// TIA Portal V16 export
// export: Created 2023-03-29T11:04:47.8257931Z, ExportSetting WithDefaults, DisplayName Totally Integrated Automation Portal, DisplayVersion V16 Update 6, DisplayName TIA Portal Version Control Interface, DisplayVersion V16 Update 2, DisplayName TIA Portal Openness, DisplayVersion V16 Update 6, DisplayName STEP 7 Professional, DisplayVersion V16 Update 6, DisplayName STEP 7 Safety, DisplayVersion V16, DisplayName WinCC Advanced, DisplayVersion V16 Update 6
FUNCTION_BLOCK "Sterowanie dołączeniem falownika"   // FB8, LAD
TITLE = Sterowanie dołączaniem styczników falownika
{ S7_Optimized_Access := 'TRUE' }
AUTHOR : rtecmer
VERSION : 0.1
// Sterowa stycznikiem pracy z falownika.
// Funkcja FB8 komutuje załaczenie stycznika FALOWNIK dla konkretnego napędu. Napędem sterowanym jest zawsze napęd przypisany do MC (czyli IsReady_MC to jest gotowość napędu sterowaniego) Na wejścia oznaczone wyróżnikiem MC podlączamy sygnały tej samej dmuchawy, której stycznikiem będziemy sterować poprzez wtjście setSUPV_FM
//  
// Sterowanie stycznikiem . Ustawianie znaczników setCMD_FM i setSUPV_FM które przekazywane są do funkcji FC3/FC1 DRV01 driver napędów. Następnie przekazywane jest do warstwy Hawtware/ OUT gdzie ustawiane jest wyjście sterownika
// stored: AutoNumber true, IsIECCheckEnabled false, IsRetainMemResEnabled false, MemoryReserve 500, SetENOAutomatically false, UDAEnableTagReadback false
   VAR_INPUT
      Is_up_Hz : Bool;
      Set_HWork_M : Bool;   // Znacznik ustawienia pracy od licznika
      setPID_Pompy : Bool;   // Znacznik załączenie, regulacji falownika
      IsRunInverter_MA : Bool;   // Potwierdzenie pracy z falownika kompresor dodatkowy 1
      IsRunNetwork_MA : Bool;   // Potwierdzenie praca z sieć dodatkowego
      IsRunInverter_MB : Bool;   // Potwierdzenie pracy z falownika kompresor dodatkowy 2
      IsRunNetwork_MB : Bool;   // Potwierdzenie praca z sieć dodatkowego
      IsRunNetwork_MC : Bool;   // Potwierdzenie pracy z sieci
      IsRunInverter_MC : Bool;   // Potwierdzenie pracy z falownika
      IsRunNetwork_MD : Bool;   // Potwierdzenie pracy z sieci
      IsRunInverter_MD : Bool;   // Potwierdzenie pracy z falownika
      FC2_Set_50H : Bool;   // Znacznik osiągnięcia czasu dla 50Hz
      IsRunInverter1 : Bool;   // Potwierdzenie pracy falownika / Potwierdzenie pracy falownika kompresorów M7M8M9
      AlwaysTRUE : Bool;
      IsReady_MA : Bool;   // Znacznik gotowości
      IsReady_MB : Bool;   // Znacznik gotowości
      IsReady_MC : Bool;   // Znacznik gotowości
      IsReady_MD : Bool;   // Znacznik gotowości
      IsModeAut : Bool;   // Znacznik trybu automat
      FB9_Set_Motor2 : Bool;   // Polecenie dostawienia dodatkowej nr1
      FB9_Set_Motor3 : Bool;   // Polecenie dostawienia dodatkowej nr2
      FB9_Set_Motor4 : Bool;   // Polecenie dostawienia dodatkowej nr3
      IsReady_Inverter : Bool;   // Gotowość falownika
      ResWorkInverter_to_MaxTime : Bool;   // Bit kasowania pracy falownika od maxymalnej ciągłej pracy
   END_VAR
   VAR_OUTPUT
      setSUPV_FM : Bool;   // Znacznik polecenia startu z falownika
   END_VAR
   VAR_IN_OUT
      setCMD_FM : Bool;   // Znacznik sterowania w trybie falownik
      Timer_OFF_Inverter_M : TOF_TIME;   // Timer na blokowanie po odłączeniu stycznika falownika
      Timer_Start_Inver_M : TON_TIME;   // Timer opóźnienia załaczenia stycznika pracy z falownika
      Timer_Set50Hz_Off_Inver_M : TON_TIME;   // Timer opóźnieniawyłączeniea falownika
      Mem_Res_setCMD_MC : Bool;   // pamięć zbocza załączenia timera blokowania stycznika falowni
   END_VAR
   VAR
      Network_50Hz : Bool;   // Znacznik 50 Hz podtrzymanie przełączenia na sieć
   END_VAR
   VAR_TEMP
      IsDrive_Optimum : Bool;   // Znacznik optymalnej ilości napędów. Jeśli False to nie przełaczaj Falowni/Sieć
      CMD_OFF_inverter : Bool;   // Wyłączenie falownika od 50Hz i dodatkowa / Wyłączenie falownika od 50Hz i udtawiona dodatkowa
      tmpOFF_inverter : Bool;
   END_VAR
   VAR_TEMP   // added for the SCL form of the ladder/FBD networks
      _w1 : Bool;
      _w2 : Bool;
   END_VAR
BEGIN

REGION Network 1: Control status motors / Kontrola statusu napędu
   // // Dostępna  jedna dmuchawa gdy wartość 1, 2, 4
   // // Dostępne dwie dmuchawy gdy wartość 6, 5, 3 
   // // Dostępne trzy dmuchawy gdy wartość 7
END_REGION

REGION Network 2: Histereza na dołączenie stycznika falownika
   // Sterowanie dołączeniem stycznika pracy z falownika
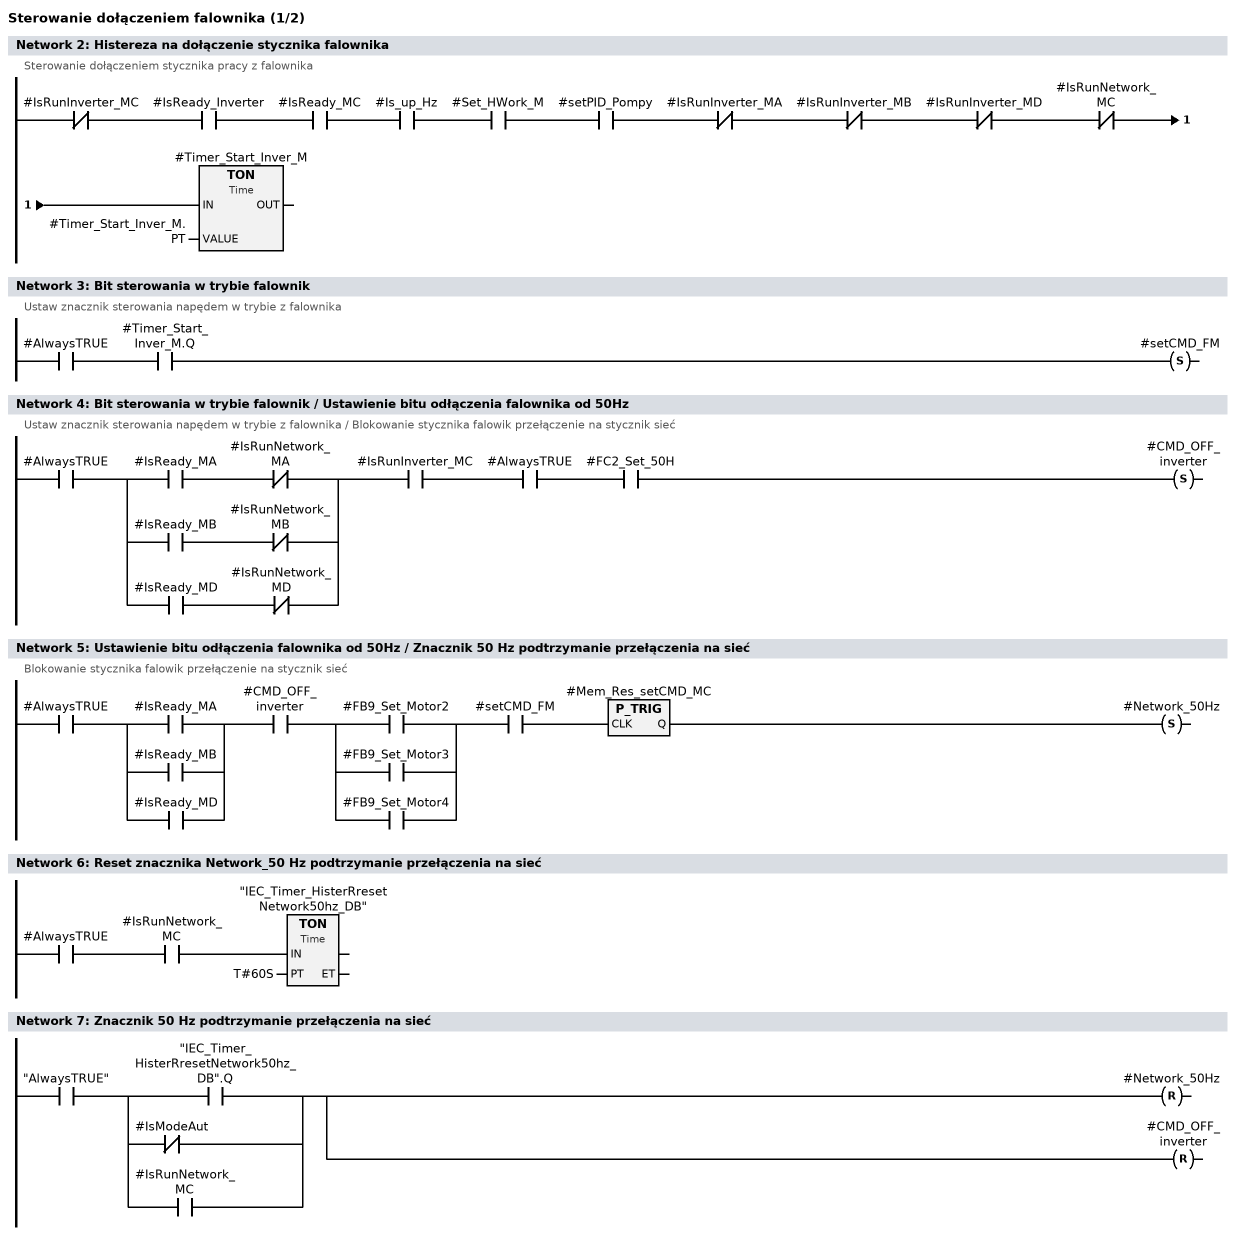
   #Timer_Start_Inver_M(IN := NOT #IsRunInverter_MC AND #IsReady_Inverter AND #IsReady_MC AND #Is_up_Hz AND #Set_HWork_M AND #setPID_Pompy AND NOT #IsRunInverter_MA AND NOT #IsRunInverter_MB AND NOT #IsRunInverter_MD AND NOT #IsRunNetwork_MC, PT := #Timer_Start_Inver_M.PT);   // TON coil
END_REGION

REGION Network 3: Bit sterowania w trybie falownik
   // Ustaw znacznik sterowania napędem w trybie z falownika
   RUNG wire#powerrail
      Contact( #AlwaysTRUE )
      Contact( #Timer_Start_Inver_M.Q )
      S_Coil( #setCMD_FM )
   END_RUNG
   // the same network as SCL:
   IF #AlwaysTRUE AND #Timer_Start_Inver_M.Q THEN #setCMD_FM := TRUE; END_IF;
END_REGION

REGION Network 4: Bit sterowania w trybie falownik / Ustawienie bitu odłączenia falownika od 50Hz
   // Ustaw znacznik sterowania napędem w trybie z falownika / Blokowanie stycznika falowik przełączenie na stycznik sieć
   RUNG wire#powerrail
      Contact( #AlwaysTRUE )
      wire#w1
      Contact( #IsReady_MA )
      I_Contact( #IsRunNetwork_MA )
      wire#w2
      Contact( #IsRunInverter_MC )
      Contact( #AlwaysTRUE )
      Contact( #FC2_Set_50H )
      S_Coil( #CMD_OFF_inverter )
   END_RUNG
   RUNG wire#w1
      Contact( #IsReady_MB )
      I_Contact( #IsRunNetwork_MB )
   END_RUNG wire#w2
   RUNG wire#w1
      Contact( #IsReady_MD )
      I_Contact( #IsRunNetwork_MD )
   END_RUNG wire#w2
   // the same network as SCL:
   IF #AlwaysTRUE AND ((#IsReady_MA AND NOT #IsRunNetwork_MA) OR (#IsReady_MB AND NOT #IsRunNetwork_MB) OR (#IsReady_MD AND NOT #IsRunNetwork_MD)) AND #IsRunInverter_MC AND #AlwaysTRUE AND #FC2_Set_50H THEN
       #CMD_OFF_inverter := TRUE;
   END_IF;
END_REGION

REGION Network 5: Ustawienie bitu odłączenia falownika od 50Hz / Znacznik 50 Hz podtrzymanie przełączenia na sieć
   // Blokowanie stycznika falowik przełączenie na stycznik sieć
   RUNG wire#powerrail
      Contact( #AlwaysTRUE )
      wire#w1
      Contact( #IsReady_MA )
      wire#w2
      Contact( #CMD_OFF_inverter )
      wire#w3
      Contact( #FB9_Set_Motor2 )
      wire#w4
      Contact( #setCMD_FM )
      P_Trig( #Mem_Res_setCMD_MC )
      S_Coil( #Network_50Hz )
   END_RUNG
   RUNG wire#w1
      Contact( #IsReady_MB )
   END_RUNG wire#w2
   RUNG wire#w1
      Contact( #IsReady_MD )
   END_RUNG wire#w2
   RUNG wire#w3
      Contact( #FB9_Set_Motor3 )
   END_RUNG wire#w4
   RUNG wire#w3
      Contact( #FB9_Set_Motor4 )
   END_RUNG wire#w4
   // the same network as SCL:
   #_w1 := #AlwaysTRUE AND (#IsReady_MA OR #IsReady_MB OR #IsReady_MD) AND #CMD_OFF_inverter AND (#FB9_Set_Motor2 OR #FB9_Set_Motor3 OR #FB9_Set_Motor4) AND #setCMD_FM;
   #_w2 := #_w1 AND NOT #Mem_Res_setCMD_MC;   // rising edge
   #Mem_Res_setCMD_MC := #_w1;
   IF #_w2 THEN #Network_50Hz := TRUE; END_IF;
END_REGION

REGION Network 6: Reset znacznika Network_50 Hz podtrzymanie przełączenia na sieć
   RUNG wire#powerrail
      Contact( #AlwaysTRUE )
      Contact( #IsRunNetwork_MC )
      { S7_Templates := "time_type := Time" } "IEC_Timer_HisterRresetNetwork50hz_DB".TON(pt := T#60S, et =>)
   END_RUNG
   // the same network as SCL:
   "IEC_Timer_HisterRresetNetwork50hz_DB".TON(IN := #AlwaysTRUE AND #IsRunNetwork_MC, PT := T#60S);
END_REGION

REGION Network 7: Znacznik 50 Hz podtrzymanie przełączenia na sieć
   RUNG wire#powerrail
      Contact( "AlwaysTRUE" )
      wire#w1
      Contact( "IEC_Timer_HisterRresetNetwork50hz_DB".Q )
      wire#w2
      R_Coil( #Network_50Hz )
   END_RUNG
   RUNG wire#w1
      I_Contact( #IsModeAut )
   END_RUNG wire#w2
   RUNG wire#w1
      Contact( #IsRunNetwork_MC )
   END_RUNG wire#w2
   RUNG wire#w2
      R_Coil( #CMD_OFF_inverter )
   END_RUNG
   // the same network as SCL:
   IF "AlwaysTRUE" AND ("IEC_Timer_HisterRresetNetwork50hz_DB".Q OR NOT #IsModeAut OR #IsRunNetwork_MC) THEN
       #Network_50Hz := FALSE;
       #CMD_OFF_inverter := FALSE;
   END_IF;
END_REGION

REGION Network 8: Timer blokowania po odłączenieu stycznika falownik
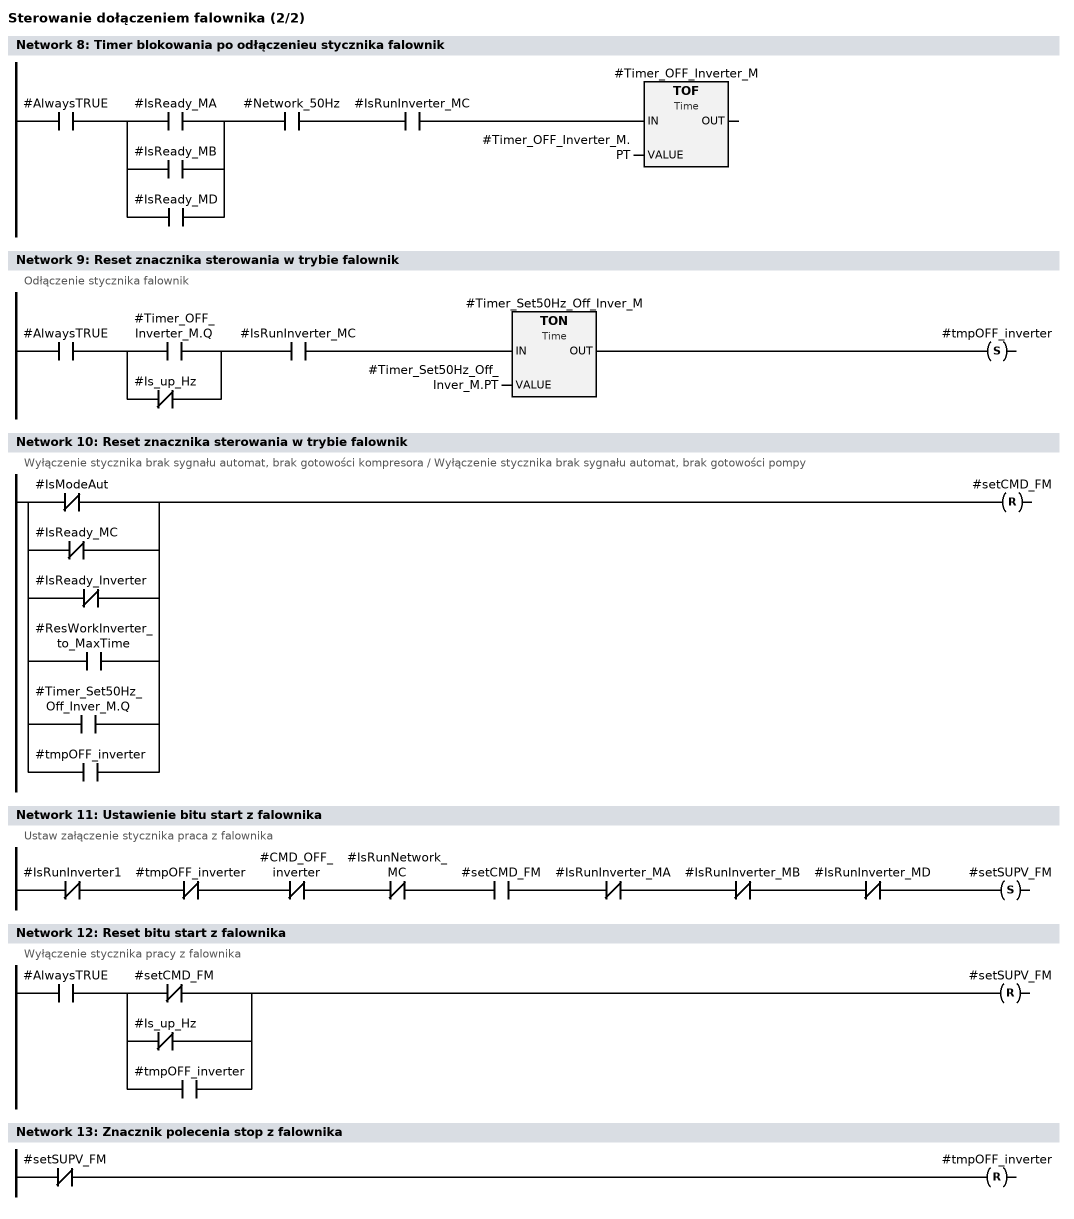
   #Timer_OFF_Inverter_M(IN := #AlwaysTRUE AND (#IsReady_MA OR #IsReady_MB OR #IsReady_MD) AND #Network_50Hz AND #IsRunInverter_MC, PT := #Timer_OFF_Inverter_M.PT);   // TOF coil
END_REGION

REGION Network 9: Reset znacznika sterowania w trybie falownik
   // Odłączenie stycznika falownik
   #_w1 := #AlwaysTRUE AND (#Timer_OFF_Inverter_M.Q OR NOT #Is_up_Hz) AND #IsRunInverter_MC;
   #Timer_Set50Hz_Off_Inver_M(IN := #_w1, PT := #Timer_Set50Hz_Off_Inver_M.PT);   // TON coil
   IF #_w1 THEN #tmpOFF_inverter := TRUE; END_IF;
END_REGION

REGION Network 10: Reset znacznika sterowania w trybie falownik
   // Wyłączenie stycznika brak sygnału automat, brak gotowości kompresora / Wyłączenie stycznika brak sygnału automat, brak gotowości pompy
   RUNG wire#powerrail
      I_Contact( #IsModeAut )
      wire#w1
      R_Coil( #setCMD_FM )
   END_RUNG
   RUNG wire#powerrail
      I_Contact( #IsReady_MC )
   END_RUNG wire#w1
   RUNG wire#powerrail
      I_Contact( #IsReady_Inverter )
   END_RUNG wire#w1
   RUNG wire#powerrail
      Contact( #ResWorkInverter_to_MaxTime )
   END_RUNG wire#w1
   RUNG wire#powerrail
      Contact( #Timer_Set50Hz_Off_Inver_M.Q )
   END_RUNG wire#w1
   RUNG wire#powerrail
      Contact( #tmpOFF_inverter )
   END_RUNG wire#w1
   // the same network as SCL:
   IF NOT #IsModeAut OR NOT #IsReady_MC OR NOT #IsReady_Inverter OR #ResWorkInverter_to_MaxTime OR #Timer_Set50Hz_Off_Inver_M.Q OR #tmpOFF_inverter THEN
       #setCMD_FM := FALSE;
   END_IF;
END_REGION

REGION Network 11: Ustawienie bitu start z falownika
   // Ustaw załączenie stycznika praca z falownika
   RUNG wire#powerrail
      I_Contact( #IsRunInverter1 )
      I_Contact( #tmpOFF_inverter )
      I_Contact( #CMD_OFF_inverter )
      I_Contact( #IsRunNetwork_MC )
      Contact( #setCMD_FM )
      I_Contact( #IsRunInverter_MA )
      I_Contact( #IsRunInverter_MB )
      I_Contact( #IsRunInverter_MD )
      S_Coil( #setSUPV_FM )
   END_RUNG
   // the same network as SCL:
   IF NOT #IsRunInverter1 AND NOT #tmpOFF_inverter AND NOT #CMD_OFF_inverter AND NOT #IsRunNetwork_MC AND #setCMD_FM AND NOT #IsRunInverter_MA AND NOT #IsRunInverter_MB AND NOT #IsRunInverter_MD THEN
       #setSUPV_FM := TRUE;
   END_IF;
END_REGION

REGION Network 12: Reset bitu start z falownika
   // Wyłączenie stycznika pracy z falownika
   RUNG wire#powerrail
      Contact( #AlwaysTRUE )
      wire#w1
      I_Contact( #setCMD_FM )
      wire#w2
      R_Coil( #setSUPV_FM )
   END_RUNG
   RUNG wire#w1
      I_Contact( #Is_up_Hz )
   END_RUNG wire#w2
   RUNG wire#w1
      Contact( #tmpOFF_inverter )
   END_RUNG wire#w2
   // the same network as SCL:
   IF #AlwaysTRUE AND (NOT #setCMD_FM OR NOT #Is_up_Hz OR #tmpOFF_inverter) THEN
       #setSUPV_FM := FALSE;
   END_IF;
END_REGION

REGION Network 13: Znacznik polecenia stop z falownika
   RUNG wire#powerrail
      I_Contact( #setSUPV_FM )
      R_Coil( #tmpOFF_inverter )
   END_RUNG
   // the same network as SCL:
   IF NOT #setSUPV_FM THEN #tmpOFF_inverter := FALSE; END_IF;
END_REGION
END_FUNCTION_BLOCK
